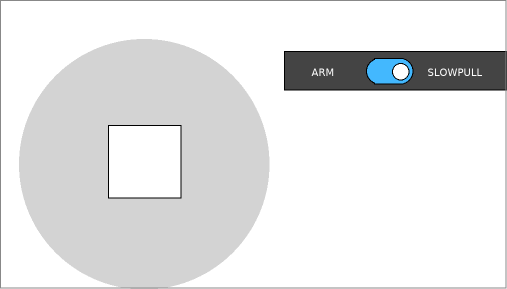
VISUALIZATION Popup_SlowpullJog  // 507x289
    Ellipse (19,39 250x250)
    RoundedRectangle (108,125 73x73)
    Group (284,51 223x42)
        RoundedRectangle (0,0 223x39)
        Label (1,1 76x41), "ARM"
        Label (128,1 86x41), "SLOWPULL"
        Group (82,7 43x26)
            OnMouseClick: toggle HMI_Ctrl.bSlowpullJogPageEnable
            Group (0,0 47x26)
                Ellipse (0,0 26x26)
                Ellipse (21,0 26x26)
                RoundedRectangle (8,0 29x26)
            Ellipse (1,1 24x24)
            Ellipse (23,1 23x24)
            RoundedRectangle (9,1 28x24)
            Ellipse (26,5 17x17)
END_VISUALIZATION

(* stored: Version 1.1.0.1, ProductVersion 3.1.4024.12
   Visu Popup_SlowpullJog: Id {2b48ad6a-7141-40ca-8e04-0df64b1e9b9b} *)
